{attribute 'qualified_only'}
{attribute 'strict'}
{attribute 'To_string'}
TYPE eNetcomState :
(
	NotConnected := 0,
	OK:=1,
	Warning:=2,
	Error:=3
);
END_TYPE

(* stored: Version 1.1.0.1, ProductVersion 3.1.4026.18
   DUT eNetcomState: Id {d261cc99-f85b-46a4-86a0-807b6fa97a11} *)
